// TwinCAT 3 PLC project VacuumSystemSimulator
// Title: Vacuum System Simulator Library
// Company: SLAC
// ProjectVersion: 0.2.10
// Description: Library of functions used for simulation of vacuum systems.
// ProgramVersion: 3.1.4020.1
// libraries:
//   VisuElem3DPath, 3.5.6.0 (System)
//   VisuElemMeter, 3.5.6.0 (System)
//   VisuElems, 3.5.6.10 (System)
//   VisuElemsDateTime, 3.5.6.0 (System)
//   VisuElemsSpecialControls, 3.5.6.0 (System)
//   VisuElemsWinControls, 3.5.6.0 (System)
//   VisuElemTextEditor, 3.5.6.0 (System)
//   visuinputs, 3.5.6.0 (system)
//   VisuNativeControl, 3.5.6.0 (System)
//   Tc2_ControllerToolbox, * (Beckhoff Automation GmbH)
//   Tc2_Standard, * (Beckhoff Automation GmbH)
//   Tc2_System, * (Beckhoff Automation GmbH)
//   Tc3_Interfaces, * (Beckhoff Automation GmbH)
//   Tc3_Module, * (Beckhoff Automation GmbH)
// project tree:
//   DUTs/ ST_CapManometer.TcDUT (not stored), ST_CapManometer_CMR362.TcDUT (not stored), ST_GAM_PIP.TcDUT, ST_MKS_317.TcDUT (not stored), ST_MKS_500.TcDUT, ST_MechPump.TcDUT (not stored), ST_MKS_275.TcDUT (not stored), ST_MKS_626.TcDUT (not stored), ST_MKS_722.TcDUT (not stored), ST_MKS_903.TcDUT (not stored), ST_MKS_907.TcDUT (not stored), ST_MKS_909.TcDUT (not stored), ST_MKS_925.TcDUT (not stored), ST_TwinScrewRoughPump.TcDUT (not stored), ST_VacuumGauge.TcDUT, ST_VacuumValve.TcDUT, ST_MKS_422.TcDUT, ST_VAT_77FS.TcDUT (not stored), ST_Volume.TcDUT (not stored)
//   GVLs/ GVL.TcGVL (not stored), GVL_VSS_CONSTANT.TcGVL (not stored)
//   POUs/ FB_Aperture.TcPOU (not stored), FB_CapManometer.TcPOU (not stored), FB_CapManometer_CMR362.TcPOU (not stored), FB_GAM_PIP.TcPOU (not stored), FB_MKS_275.TcPOU (not stored), FB_MKS_275_to_500_HvOn.TcPOU (not stored), FB_MKS_422.TcPOU (not stored), FB_MKS_500.TcPOU, FB_MKS_907.TcPOU (not stored), FB_MKS_909.TcPOU (not stored), FB_MKS_903.TcPOU (not stored), FB_MKS_925.TcPOU (not stored), FB_RoughPump_Demo.TcPOU (not stored) (excluded from build), FB_SetChamberPressure.TcPOU (not stored), FB_TurboPump.TcPOU (not stored), FB_RoughPump.TcPOU (not stored), FB_PfeifferTurboPump.TcPOU (not stored) (excluded from build), FB_TurboPump_Demo.TcPOU (not stored) (excluded from build), FB_VacuumValve_old.TcPOU (not stored) (excluded from build), FB_VacuumValve.TcPOU (not stored), FB_VacuumValve_Vent.TcPOU (not stored), FB_VirtualLeak.TcPOU (not stored)
//   POUs/VacuumGaugePressureFunctions/ F_MKS_907.TcPOU (not stored) (excluded from build), F_MKS_903.TcPOU (not stored) (excluded from build), F_MKS_925.TcPOU (not stored) (excluded from build), F_MKS_937.TcPOU (not stored), F_MKS_500.TcPOU (not stored) (excluded from build), F_MKS_275.TcPOU (not stored) (excluded from build), F_MKS_909.TcPOU (not stored) (excluded from build)
//   Version/ Global_Version.TcGVL (not stored)
//   VISUs/ Main.TcVIS (not stored)

// ---- DUTs/ST_GAM_PIP.TcDUT
TYPE ST_GAM_PIP :
STRUCT
	//Discrete Readback 
	xOn AT%I*:BOOL; //Readback of whether Gamma Ion Pump is turned on or not
END_STRUCT
END_TYPE

// ---- DUTs/ST_MKS_500.TcDUT
TYPE ST_MKS_500 EXTENDS ST_VacuumGauge :
STRUCT
	//Discrete Control: Ion gauges only
	i_xHvOn	 AT%I*:BOOL	; //High voltage On to turn on this Cold Cathode gauge
	q_xHVOn AT%Q*:BOOL ;
	q_DisActive AT%Q*:BOOL ;
	// Simulation parameters
	tonIC	:	TON := (PT := T#10S);// takes 10 seconds to turn on this Cold Cathode gauge
END_STRUCT
END_TYPE

// ---- DUTs/ST_VacuumGauge.TcDUT
TYPE ST_VacuumGauge :
STRUCT
	(* Simulation parameters *)
	rPress	:	REAL;//The real pressure coming from the ST_volume @ a chamber
	
	(* IO Readback *)
	q_iRawPress	 AT%Q*:	INT;// The transformed integer from real pressure to an integer encoded signal to be passed to the PLC 
	
	(* Testing Connection *)
	q_xGaugeConnected	: BOOL;// to connect and disconnect gauge, easy to check whether gauge in connected at correct location

END_STRUCT
END_TYPE

// ---- DUTs/ST_VacuumValve.TcDUT
TYPE ST_VacuumValve :
STRUCT

	//Discrete controls
	i_xSol	 AT%I*	:BOOL;//Solenoid to control the valve( either closed or open)
	
	//Discrete readbacks
	q_xOpnLS  AT%Q*: BOOL;//readback whether open
	q_xClsLS  AT%Q*: BOOL;//readback whether closed
END_STRUCT
END_TYPE

// ---- DUTs/ST_MKS_422.TcDUT
TYPE ST_MKS_422 EXTENDS ST_VacuumGauge :
STRUCT
	
	//Discrete Control: Ion gauges only
	i_xHvOn	 AT%I*:	BOOL;//High voltage On to turn on ion gauges
	
	// Simulation parameters
	tonIC	:	TON := (PT := T#10S);// takes 10 seconds to turn on this gauge
END_STRUCT
END_TYPE

// ---- POUs/FB_MKS_500.TcPOU
FUNCTION_BLOCK FB_MKS_500
VAR_INPUT
	stVolume : ST_Volume;
END_VAR
VAR_OUTPUT
END_VAR
VAR_IN_OUT
	stGauge	:	ST_MKS_500;
END_VAR
VAR
END_VAR
VAR CONSTANT
END_VAR

(* 
MKS 500 Vacuum gauge

A vacuum gauge takes as input, the pressure of the volume it is attached to,
and produces on its analog output, a corresponding voltage.

A.Pai
3/29/2017
*)

(* Operation 
When the HV on signal is active, the gauge will take a little bit of time to
start an ion current.
*)
stGauge.tonIC.IN	:=	stGauge.i_xHvOn;	
stGauge.tonIC();

stGauge.rPress := stVolume.rPressure; //always this because we assume the gauge is actually physically connected

IF stGauge.q_xGaugeConnected THEN//If gauge is connected
	
	stGauge.q_iRawPress := M_MKS_500(
	i_rPress := stGauge.rPress,
	i_xHVOn	:=	stGauge.i_xHvOn,
	i_xICOn	:=	stGauge.tonIC.Q
	);// gauge on
	
	
	stGauge.i_xHvOn := TRUE;
	IF (stGauge.q_iRawPress = 0.5) THEN 
		stGauge.q_DisActive := FALSE; 
		stGauge.q_xHVOn := TRUE;
	ELSIF ( stGauge.q_iRawPress = 0.1) THEN
		stGauge.q_DisActive := FALSE; 
		stGauge.q_xHVOn := FALSE;
	ELSE 
		stGauge.q_DisActive := TRUE; 
		stGauge.q_xHVOn := TRUE;
	END_IF;

ELSE//gauge gets disconnected

	stGauge.rPress := 0;
	stGauge.q_iRawPress := 0; // gauge disconnected
	stGauge.q_xHVOn := FALSE;
	stGauge.i_xHvOn := FALSE;
	stGauge.q_DisActive := FALSE;
END_IF

METHOD PRIVATE M_MKS_500 : INT
VAR_INPUT
	i_rPress	:	REAL;
	i_xHVOn	:	BOOL;
	i_xICOn	:	BOOL;
END_VAR
VAR
	rVoltage	:	REAL;
END_VAR
VAR CONSTANT
	vBase	:	REAL := 0; //corresponding vbase 0V based on default curve.  See manual pg. 44
	pBase	:	REAL := 1.0E-10; //default curve base pressure is 1E-10. Confusing since can't actually read that low using analog out.
	vSlope	:	REAL := 1.0; //looks correct for default curve
	vNoIC	:	REAL := 0.5;
	vNoHV	:	REAL := 0.1;
END_VAR
(*
MKS 500 voltage calculation

Does the inverse of the FB 500 from the vacuum library.

A. Wallace, 2016-2-22
*)
IF i_xHVOn and i_xICOn THEN
	rVoltage := MAX(vBase, (vBase + vSlope * LOG(i_rPress/pBase)));
ELSIF i_xHVOn AND NOT i_xICOn THEN
	rVoltage := vNoIC;
ELSE
	rVoltage := vNoHV;
END_IF

M_MKS_500 := REAL_TO_INT( rVoltage * 32767/10 );
END_METHOD

END_FUNCTION_BLOCK
